{attribute 'Tc2GvlVarNames'}
{attribute 'strict'}
(* Stato Prodotto Nel Pick Point *)
TYPE e_Stato_Prodotto_Su_PickPoint :
(
	WORKPICKPOINT_PRODOTTO_ASSENTE	 := 0,	(* Prodotto Presente Nel PickPoint *)
	WORKPICKPOINT_PRODOTTO_PRESENTE	 := 1	(* Prodotto Assente Nel PickPoint *)
);
END_TYPE

(* stored: Version 1.1.0.1, ProductVersion 3.1.4024.11
   EnumerationTextList e_Stato_Prodotto_Su_PickPoint: Id {711c8d10-6f0f-4288-a332-a7c24decb955} *)
